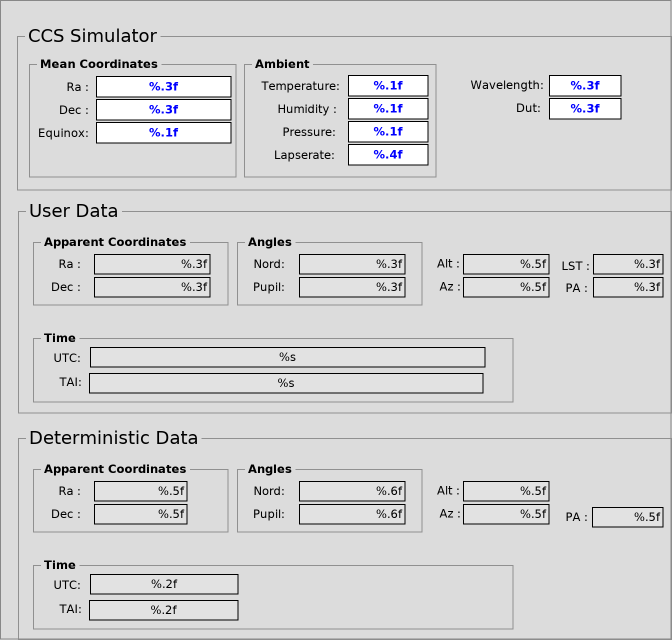
VISUALIZATION GUI_TEMPLATE_CCS_SIM  // 672x640
VAR_INPUT
	m_DeviceName : STRING;
END_VAR
VAR_IN_OUT
	m_Instance : FB_CCS_SIM;
END_VAR
    GroupBox (17,28 655x162), "CCS Simulator"
        GroupBox (12,28 207x121), "Mean Coordinates"
            Label (23,21 40x20), "Ra :"
            Label (23,44 40x20), "Dec :"
            Rectangle (67,20 135x21), "%.3f", tooltip "Mean Right Ascension [hhmmss]", text variable: m_Instance.ctrl.meanCoordinates.alpha
                OnMouseDown: write the text variable via Edit
            Rectangle (67,43 135x21), "%.3f", tooltip "Mean Declination [ddmmss]", text variable: m_Instance.ctrl.meanCoordinates.delta
                OnMouseDown: write the text variable via Edit
            Rectangle (67,66 135x21), "%.1f", tooltip "Equinox", text variable: m_Instance.ctrl.meanCoordinates.equinox
                OnMouseDown: write the text variable via Edit
            Label (3,67 60x20), "Equinox:"
        GroupBox (227,28 192x121), "Ambient"
            Label (7,20 92x20), "Temperature:"
            Label (17,43 79x20), "Humidity :"
            Rectangle (104,19 80x21), "%.1f", tooltip "Temperature [degC]", text variable: m_Instance.ctrl.environment.temperature
                OnMouseDown: write the text variable via Edit
            Rectangle (104,42 80x21), "%.1f", tooltip "Humidity [%]", text variable: m_Instance.ctrl.environment.humidity
                OnMouseDown: write the text variable via Edit
            Rectangle (104,65 80x21), "%.1f", tooltip "Pressure [mbar]", text variable: m_Instance.ctrl.environment.pressure
                OnMouseDown: write the text variable via Edit
            Label (25,66 70x20), "Pressure:"
            Label (24,89 70x20), "Lapserate:"
            Rectangle (104,88 80x21), "%.4f", tooltip "Lapse Rate", text variable: m_Instance.ctrl.environment.lapserate
                OnMouseDown: write the text variable via Edit
        Rectangle (532,47 72x21), "%.3f", text variable: m_Instance.ctrl.wavelength
            OnMouseDown: write the text variable via Edit
        Rectangle (532,70 72x21), "%.3f", text variable: m_Instance.ctrl.dut
            OnMouseDown: write the text variable via Edit
        Label (481,70 46x20), "Dut:"
    GroupBox (18,203 654x210), "User Data"
        GroupBox (15,31 195x71), "Apparent Coordinates"
            Label (11,20 40x20), "Ra :"
            Label (11,43 40x20), "Dec :"
            Label (8,70 60x20)
            Rectangle (61,43 116x20), "%.3f", tooltip "Apparent Declination [ddmmss]", text variable: m_Instance.stat.gui_data.dec
            Rectangle (61,20 116x20), "%.3f", tooltip "Apparent Right Ascension [hhmmss]", text variable: m_Instance.stat.gui_data.ra
        Rectangle (575,74 70x20), "%.3f", tooltip "Parallactic Angle [deg]", text variable: m_Instance.stat.gui_data.pa
        Label (523,75 50x20), "PA :"
        Label (408,51 37x19), "Alt :"
        Label (411,74 35x19), "Az :"
        GroupBox (219,31 185x71), "Angles"
            Label (11,20 40x20), "Nord:"
            Label (11,43 40x20), "Pupil:"
            Label (8,70 60x20)
            Rectangle (62,20 106x20), "%.3f", tooltip "North angle [deg]", text variable: m_Instance.stat.gui_data.north_angle
            Rectangle (62,43 106x20), "%.3f", tooltip "Pupil angle[deg]", text variable: m_Instance.stat.gui_data.pupil_angle
        Rectangle (445,74 86x20), "%.5f", tooltip "TEL Azimuth [deg]", text variable: m_Instance.stat.gui_data.az
        Rectangle (445,51 86x20), "%.5f", tooltip "TEL Altitude [deg]", text variable: m_Instance.stat.gui_data.alt
        GroupBox (15,127 480x72), "Time"
            Label (11,18 40x20), "UTC:"
            Label (6,42 46x20), "TAI:"
            Label (8,70 60x20)
            Rectangle (57,17 395x20), "%s", tooltip "UTC time [sec]", text variable: m_Instance.refTimeObj.stat.sUtcTime
            Rectangle (56,43 394x20), "%s", tooltip "TAI time [sec]", text variable: m_Instance.refTimeObj.stat.sTaiTime
    Label (464,75 83x20), "Wavelength:"
    Label (552,256 41x20), "LST :"
    Rectangle (593,254 70x20), "%.3f", tooltip "Local Sidereal Time [h]", text variable: m_Instance.stat.gui_data.lst
    GroupBox (18,430 654x210), "Deterministic Data"
        GroupBox (15,31 195x71), "Apparent Coordinates"
            Label (11,20 40x20), "Ra :"
            Label (11,43 40x20), "Dec :"
            Label (8,70 60x20)
            Rectangle (61,43 93x20), "%.5f", tooltip "Apparent Declination [rad]", text variable: m_Instance.stat.data.radec_at_altaz_at_requested_xy[1]
            Rectangle (61,20 93x20), "%.5f", tooltip "Apparent Right Ascension [rad]", text variable: m_Instance.stat.data.radec_at_altaz_at_requested_xy[0]
        Rectangle (574,77 71x20), "%.5f", tooltip "Parallactic Angle [rad]", text variable: m_Instance.stat.data.parallactic_angle
        Label (523,77 50x20), "PA :"
        Label (408,51 37x19), "Alt :"
        Label (411,74 35x19), "Az :"
        GroupBox (219,31 185x71), "Angles"
            Label (11,20 40x20), "Nord:"
            Label (11,43 40x20), "Pupil:"
            Label (8,70 60x20)
            Rectangle (62,20 106x20), "%.6f", tooltip "North angle [rad]", text variable: m_Instance.stat.data.north_angle
            Rectangle (62,43 106x20), "%.6f", tooltip "Pupil angle[rad]", text variable: m_Instance.stat.data.pupil_angle
        Rectangle (445,74 86x20), "%.5f", tooltip "TEL Azimuth [rad]", text variable: m_Instance.stat.data.current_observed_altaz[1]
        Rectangle (445,51 86x20), "%.5f", tooltip "TEL Altitude [rad]", text variable: m_Instance.stat.data.current_observed_altaz[0]
        GroupBox (15,127 480x72), "Time"
            Label (11,18 40x20), "UTC:"
            Label (6,42 46x20), "TAI:"
            Label (8,70 60x20)
            Rectangle (57,17 148x20), "%.2f", tooltip "UTC time [sec]", text variable: m_Instance.stat.data.time_utc
            Rectangle (56,43 149x20), "%.2f", tooltip "TAI time [sec]", text variable: m_Instance.stat.data.time_tai
END_VISUALIZATION

(* stored: Version 1.1.0.1, ProductVersion 3.1.4024.11
   Visu GUI_TEMPLATE_CCS_SIM: Id {f233d3d3-a08f-4bf9-918e-57222bcffbb9} *)
